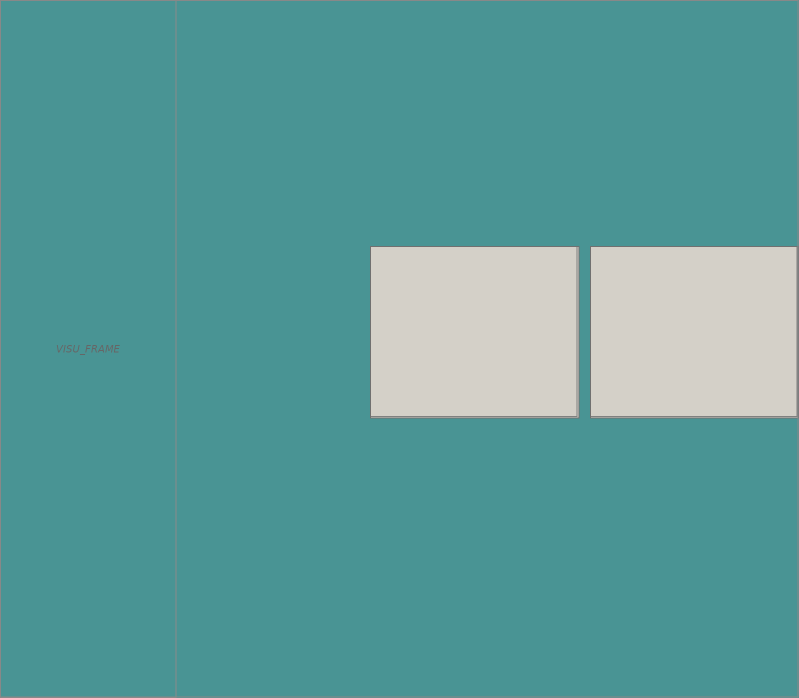
VISUALIZATION Visualization_2  // 799x698
    Button (370,246 209x172), text list: 'TextList', text index: 4
        OnMouseClick: ChangeLanguage ChangeLanguage=Türkçe
    Button (590,246 209x172), text list: 'TextList', text index: 3
        OnMouseClick: ChangeLanguage ChangeLanguage=İngilizce
    Frame (0,0 176x698)
        shows VISU_FRAME(sDayTime := MAIN.DMY_LocalTime, sTime := MAIN.HMS_LocalTime)
END_VISUALIZATION

(* stored: Version 1.1.0.1, ProductVersion 3.1.4024.4
   Visu Visualization_2: Id {2bca0815-c95d-49ec-98e1-b4149f19c27d} *)
